PROGRAM MAIN
VAR
END_VAR

END_PROGRAM

(* stored: Version 1.1.0.1
   POU MAIN: Id {76697d28-d3c1-403a-9557-5d539ac02c2d} *)
